FUNCTION_BLOCK FB_UPS_STUB IMPLEMENTS iUPS
VAR_INPUT
END_VAR
VAR_OUTPUT
END_VAR
VAR
	eUPSState :E_UPSState;
	tShutdownDelay	: TIME := T#5S;
	test_timer :Tc2_Standard.TON;
END_VAR

{warning 'add method implementation '}
METHOD persist_data : BOOL
END_METHOD

{warning 'add method implementation '}
METHOD shutdown : BOOL
END_METHOD

{warning 'add property implementation'}
PROPERTY shutdown_delay : TIME
GET
shutdown_delay := tShutdownDelay;
END_GET
SET
tShutdownDelay := shutdown_delay;
END_SET
END_PROPERTY

{warning 'add property implementation'}
PROPERTY UPSState : E_UPSState
GET
UPSState := eUPSState;
END_GET
END_PROPERTY

{warning 'add method implementation '}
METHOD watch_status : BOOL
IF eUPSState = E_UPSState.on_battery THEN
	test_timer.PT := tShutdownDelay;
ELSE
	test_timer.PT := T#15S;
END_IF

test_timer(IN := NOT test_timer.Q);

IF test_timer.Q THEN
	CASE eUPSState OF
		E_UPSState.init:
			eUPSState := E_UPSState.on_power;
		E_UPSState.on_power:
			eUPSState := E_UPSState.on_battery;
		E_UPSState.critical_error:
			eUPSState := E_UPSState.init;
	END_CASE
END_IF
END_METHOD

END_FUNCTION_BLOCK

(* stored: Version 1.1.0.1, ProductVersion 3.1.4024.12
   POU FB_UPS_STUB: Id {f8beab30-01cc-40c7-b2a7-658d7ed595f1}, SpecialFunc None
   Method persist_data: Id {31b2e3b0-a301-4fff-b03d-315c1277bef7}
   Method shutdown: Id {7b89aabf-1f3d-4f04-afa9-98f1042fbc14}
   Property shutdown_delay: Id {2b1f82ec-e073-472f-a673-cac9ec23088e}
   Get Get: Id {a264f190-c91a-4a51-bf4b-824389fe71aa}
   Set Set: Id {4777ceaf-18ca-4933-8f7d-293894b8d609}
   Property UPSState: Id {54b7a120-7be4-40bb-9128-9de12244ea4b}
   Get Get: Id {8bfda4c0-467b-45b4-8d53-7fd29aeeb8cd}
   Method watch_status: Id {a9c88e17-4cde-46fc-a941-dc36c9ca2fc7} *)
